(* IEC 61131-3 sources: eCockpitGit/test_project/src/%F%00 Library/%F%JSON/%POU%FB_JSONWriter/%F%Structure/%PRO%maxSize, 1 file *)

(* ---- %GETSET%Get.st ---- *)
//This gets the amount of bytes in the buffer
// | 1         | NSN      | 22-06-20 | Creation
VAR
END_VAR

(*%!%__DELIMITER__%!%*)
maxSize		:=		bufferMaxADR - bufferAddress;
